FUNCTION_BLOCK ColorDetect
  (* Standard: 61499-2 *)
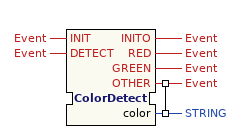
  EVENT_INPUT
    INIT;
    DETECT;
  END_EVENT
  EVENT_OUTPUT
    INITO;
    RED;
    GREEN;
    OTHER WITH color;
  END_EVENT
  VAR_OUTPUT
    color : STRING;
  END_VAR
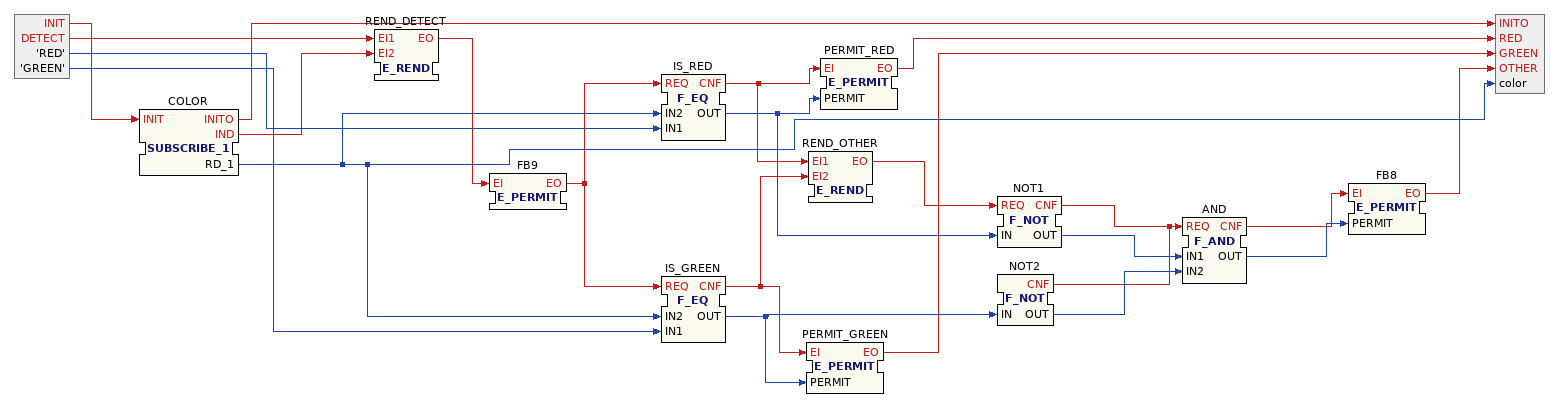
  FBS
    COLOR : SUBSCRIBE_1;
    IS_RED : F_EQ;
    IS_GREEN : F_EQ;
    AND : F_AND;
    REND_OTHER : E_REND;
    PERMIT_RED : E_PERMIT;
    PERMIT_GREEN : E_PERMIT;
    FB8 : E_PERMIT;
    FB9 : E_PERMIT;
    NOT1 : F_NOT;
    NOT2 : F_NOT;
    REND_DETECT : E_REND;
  END_FBS
  EVENT_CONNECTIONS
    COLOR.INITO TO INITO;
    INIT TO COLOR.INIT;
    FB9.EO TO IS_RED.REQ;
    FB9.EO TO IS_GREEN.REQ;
    IS_RED.CNF TO REND_OTHER.EI1;
    IS_GREEN.CNF TO REND_OTHER.EI2;
    REND_OTHER.EO TO NOT1.REQ;
    IS_RED.CNF TO PERMIT_RED.EI;
    PERMIT_RED.EO TO RED;
    IS_GREEN.CNF TO PERMIT_GREEN.EI;
    PERMIT_GREEN.EO TO GREEN;
    AND.CNF TO FB8.EI;
    FB8.EO TO OTHER;
    NOT1.CNF TO AND.REQ;
    NOT2.CNF TO AND.REQ;
    DETECT TO REND_DETECT.EI1;
    REND_DETECT.EO TO FB9.EI;
    COLOR.IND TO REND_DETECT.EI2;
  END_CONNECTIONS
  DATA_CONNECTIONS
    COLOR.RD_1 TO color;
    COLOR.RD_1 TO IS_RED.IN2;
    COLOR.RD_1 TO IS_GREEN.IN2;
    IS_RED.OUT TO NOT1.IN;
    IS_GREEN.OUT TO NOT2.IN;
    IS_RED.OUT TO PERMIT_RED.PERMIT;
    IS_GREEN.OUT TO PERMIT_GREEN.PERMIT;
    AND.OUT TO FB8.PERMIT;
    'RED' TO IS_RED.IN1;
    'GREEN' TO IS_GREEN.IN1;
    NOT1.OUT TO AND.IN1;
    NOT2.OUT TO AND.IN2;
  END_CONNECTIONS
END_FUNCTION_BLOCK
